# EPICS substitutions: CryoControlApp/Db/wcmp_misc.substitutions
file 1wcmp_misc.vdb
{
         pattern { PLC_NAME            , AREA     , LOCA , CMPNUM }
                 { PLC_CP$(CP)2_CR1$(C), CP$(CP)2 , 1$(C),   4    }
}
